FUNCTION_BLOCK BoxRingBuffer EXTENDS RingBuffer
VAR
  _bufferPtr : POINTER TO Box;  
END_VAR
VAR_STAT
  BoxId : INT := 1;
END_VAR

METHOD Append
VAR
  i : DINT;
END_VAR
i := IndexOfNextItem();

_bufferPtr[i].BoxId := THIS^.BoxId;
_bufferPtr[i].DetectedAt := ZModuleProgram.Datetime.UnixTimestamp();
_bufferPtr[i].CompletionRatio := 0;

AppendIndex();

THIS^.BoxId := THIS^.BoxId + 1;
IF THIS^.BoxId > 999
THEN
  THIS^.BoxId := 1;
END_IF
END_METHOD

/// Initializes the RingBuffer at construction time of the object by providing the bufferSize.
/// It also inidializes the pointers of head and tail with an internally stored variable.
METHOD FB_init : BOOL
VAR_INPUT
  bInitRetains : BOOL; //< if TRUE, the retain variables are initialized (warm start / cold start)
  bInCopyCode : BOOL; //< if TRUE, the instance afterwards gets moved into the copy code (online change)
  bufferSize : DINT; //< size of the **managable** buffer. The actual databuffer needs to be one element larger than bufferSize, i.e. data : ARRAY[0..bufferSize] OF ???
  bufferPtr : POINTER TO Box;
END_VAR
_bufferPtr := bufferPtr;
END_METHOD

METHOD Front : REFERENCE TO Box
VAR_INPUT
END_VAR
IF NOT THIS^.Empty
THEN
  Front REF= _bufferPtr[THIS^.IndexOfFirstItem()];
END_IF
END_METHOD

END_FUNCTION_BLOCK

(* stored: Version 1.1.0.1
   POU BoxRingBuffer: Id {4a99f8b2-47b9-47d6-8ec1-a67fc347ff72}, SpecialFunc None
   Method Append: Id {a8e942af-e8e2-43cd-9904-1704637c88bd}
   Method FB_init: Id {b7be1ef1-03c7-4484-8c4f-226576c37026}
   Method Front: Id {e4dfb401-69ee-4441-8f06-4c28e27b76c8} *)
